Staubli VAL3: onF1Event.pgx

program onF1Event()
  local num l_nFrame
  local string l_sEvent
begin
  // look if the bButton is enable
  if bButton[0] and nFrame>0
    // teach the frame
    call setPointFrame(saveData:fFrameItem[nFrame].fFrame.trsf,nFrame)
    // release
    call use:nullKey(nKey)
    use:bUseRefresh=true
  endIf
end
